(* Logix 5000 project; controller Good_Foods_96985_10252022_1208 vendor 1 type 14 code 151 rev 32.15; software revision 32.04; part 2 of 4 *)
(* tags used below, declared in another part *)
   Active_Container_Recipe : Container_Recipe;
   bAccess_Allowed : BOOL;
   bAccess_Not_Allowed : BOOL;
   bActive_Cleanout_Mode : BOOL;
   bAlwaysOff : BOOL;
   bFault_Active : BOOL;
   bHMI_PB_Left_Denester_Enabled : BOOL;
   bHMI_PB_Left_DropGate_EXT : BOOL;
   bHMI_PB_Left_DropGate_RET : BOOL;
   bHMI_PB_Left_Shuttle_EXT : BOOL;
   bHMI_PB_Left_Shuttle_RET : BOOL;
   bHMI_PB_Load_Recipe : BOOL;
   bHMI_PB_Right_Denester_Enabled : BOOL;
   bHMI_PB_Right_DropGate_EXT : BOOL;
   bHMI_PB_Right_DropGate_RET : BOOL;
   bHMI_PB_Right_Shuttle_EXT : BOOL;
   bHMI_PB_Right_Shuttle_RET : BOOL;
   bHMI_PB_Save_Recipe : BOOL;
   bHmi_PB_Set_Encoder_Home_Position : BOOL;
   bHome_1 : BOOL;
   bHome_Master_Encoder : BOOL;
   bHoming_Cmplt : BOOL;
   bHoming_Step_1 : BOOL;
   bLeft_Indexing : BOOL;
   bLeft_System_Not_Running : BOOL;
   bLeftConvBacklog_OK : BOOL;
   bLeftDropBacklog_OK : BOOL;
   bLeftPrimeBacklog_OK : BOOL;
   bLeftShuttleBacklog_OK : BOOL;
   bMaster_Encoder_Homed_After_Restart : BOOL;
   bRight_Indexing : BOOL;
   bRight_System_Not_Running : BOOL;
   bRightConvBacklog_OK : BOOL;
   bRightDropBacklog_OK : BOOL;
   bRightPrimeBacklog_OK : BOOL;
   bRightShuttleBacklog_OK : BOOL;
   bSystem_Active : BOOL;
   bSystem_Needs_To_Be_Homed : BOOL;
   Cmplt_Homing_Step_1 : BOOL;
   Container_Recipe : Container_Recipe[32];
   ctuInitLeftCyl : COUNTER;
   ctuInitRightCyl : COUNTER;   // Wont Repeat Initilation Sequence If Cmplt
   dAlarms : DINT[8];
   dHoming_Count : DINT;
   DI_PE_Left_Conv_Backlog_Present : BOOL;
   DI_PE_Left_Denest_Prime_OK : BOOL;
   DI_PE_Left_Drop_Cont_Present : BOOL;
   DI_PE_Left_Shuttle_Backlog_Present : BOOL;
   DI_PE_Right_Conv_Backlog_Present : BOOL;
   DI_PE_Right_Denest_Prime_OK : BOOL;
   DI_PE_Right_Drop_Cont_Present : BOOL;
   DI_PE_Right_Shuttle_Backlog_Present : BOOL;
   DI_PRX_Left_DropGate_EXT : BOOL;
   DI_PRX_Left_DropGate_RET : BOOL;
   DI_PRX_Left_Shuttle_RET : BOOL;
   DI_PRX_LugChain_HomingProx : BOOL;
   DI_PRX_Right_DropGate_EXT : BOOL;
   DI_PRX_Right_DropGate_RET : BOOL;
   DI_PRX_Right_Shuttle_RET : BOOL;
   dLeft_Shuttle_Seq_CMD : DINT;
   dLeft_Shuttle_Seq_CMPLT : DINT;
   DO_SOL_Left_DropGate_EXT : BOOL;
   DO_SOL_Left_DropGate_RET : BOOL;
   DO_SOL_Left_Shuttle_EXT : BOOL;
   DO_SOL_Left_Shuttle_RET : BOOL;
   DO_SOL_Right_DropGate_EXT : BOOL;
   DO_SOL_Right_DropGate_RET : BOOL;
   DO_SOL_Right_Shuttle_EXT : BOOL;
   DO_SOL_Right_Shuttle_RET : BOOL;
   dRight_Shuttle_Seq_CMD : DINT;
   dRight_Shuttle_Seq_CMPLT : DINT;
   dSystem_Start_Seq_CMPLT : DINT;
   dSystem_Stop_Seq_CMPLT : DINT;
   intHMI_RecipeListPntr : INT;
   intRecipePntr : INT;
   Left_Rev_Count : INT;
   LugChain_HomingProx_ONS : BOOL;
   LugChain_ONS_Rising : BOOL;
   mamAxisLeftSCREW_INDEXMOVE : MOTION_INSTRUCTION;
   mamAxisRightSCREW_INDEXMOVE : MOTION_INSTRUCTION;
   Master_Encoder : AXIS_CIP_DRIVE;
   ONS : DINT[16];
   rHMI_Drop_Position_Save : REAL;
   rHMI_Index_Speed_Save : REAL;
   rHMI_LefPrime_Backlog_Start_Time_S : REAL;
   rHMI_Left_Denester_Park_Pos_Save : REAL;
   rHMI_LeftConv_Backlog_Start_Time_S : REAL;
   rHMI_LeftConv_Backlog_Stop_Time_S : REAL;
   rHMI_LeftDrop_Backlog_Start_Time_S : REAL;
   rHMI_LeftDrop_Backlog_Stop_Time_S : REAL;
   rHMI_LeftPrime_Backlog_Stop_Time_S : REAL;
   rHMI_LeftShuttle_Backlog_Start_Time_S : REAL;
   rHMI_LeftShuttle_Backlog_Stop_Time_S : REAL;
   rHMI_Right_Denester_Park_Pos_Save : REAL;
   rHMI_RightConv_Backlog_Start_Time_S : REAL;
   rHMI_RightConv_Backlog_Stop_Time_S : REAL;
   rHMI_RightDrop_Backlog_Start_Time_S : REAL;
   rHMI_RightDrop_Backlog_Stop_Time_S : REAL;
   rHMI_RightPrime_Backlog_Start_Time_S : REAL;
   rHMI_RightPrime_Backlog_Stop_Time_S : REAL;
   rHMI_RightShuttle_Backlog_Start_Time_S : REAL;
   rHMI_RightShuttle_Backlog_Stop_Time_S : REAL;
   rHome_Encoder_High_Limit : REAL;
   rHome_Encoder_Low_Limit : REAL;
   Right_Rev_Count : INT;
   rSIKO_Rail_Position_Save : REAL;
   strEmpty_String : STRING;
   strHMI_Current_User : STRING;
   String : STRING;
   strMaint_String : STRING;
   strMCHS_String : STRING;
   tLeftConv_Backlog_Start : TIMER;
   tLeftConv_Backlog_Stop : TIMER;
   tLeftDrop_Backlog_Start : TIMER;
   tLeftDrop_Backlog_Stop : TIMER;
   tLeftExtDrpDly : TIMER;
   tLeftExtShutDly : TIMER;
   tLeftPrime_Backlog_Start : TIMER;
   tLeftPrime_Backlog_Stop : TIMER;
   tLeftRetDrpDly : TIMER;
   tLeftRetShutDly : TIMER;
   tLeftShuttle_Backlog_Start : TIMER;
   tLeftShuttle_Backlog_Stop : TIMER;
   tRightConv_Backlog_Start : TIMER;
   tRightConv_Backlog_Stop : TIMER;
   tRightDrop_Backlog_Start : TIMER;
   tRightDrop_Backlog_Stop : TIMER;
   tRightExtDrpDly : TIMER;
   tRightExtShutDly : TIMER;
   tRightPrime_Backlog_Start : TIMER;
   tRightPrime_Backlog_Stop : TIMER;
   tRightRetDrpDly : TIMER;
   tRightRetShutDly : TIMER;
   tRightShuttle_Backlog_Start : TIMER;
   tRightShuttle_Backlog_Stop : TIMER;
   tRightStopPosDly : TIMER;
   tRightStopPosTimeOut : TIMER;
   tTimer_Homing : TIMER;
(* MainProgram, continued *)

ROUTINE _11_Left_Shuttle_Control   (* ladder *)
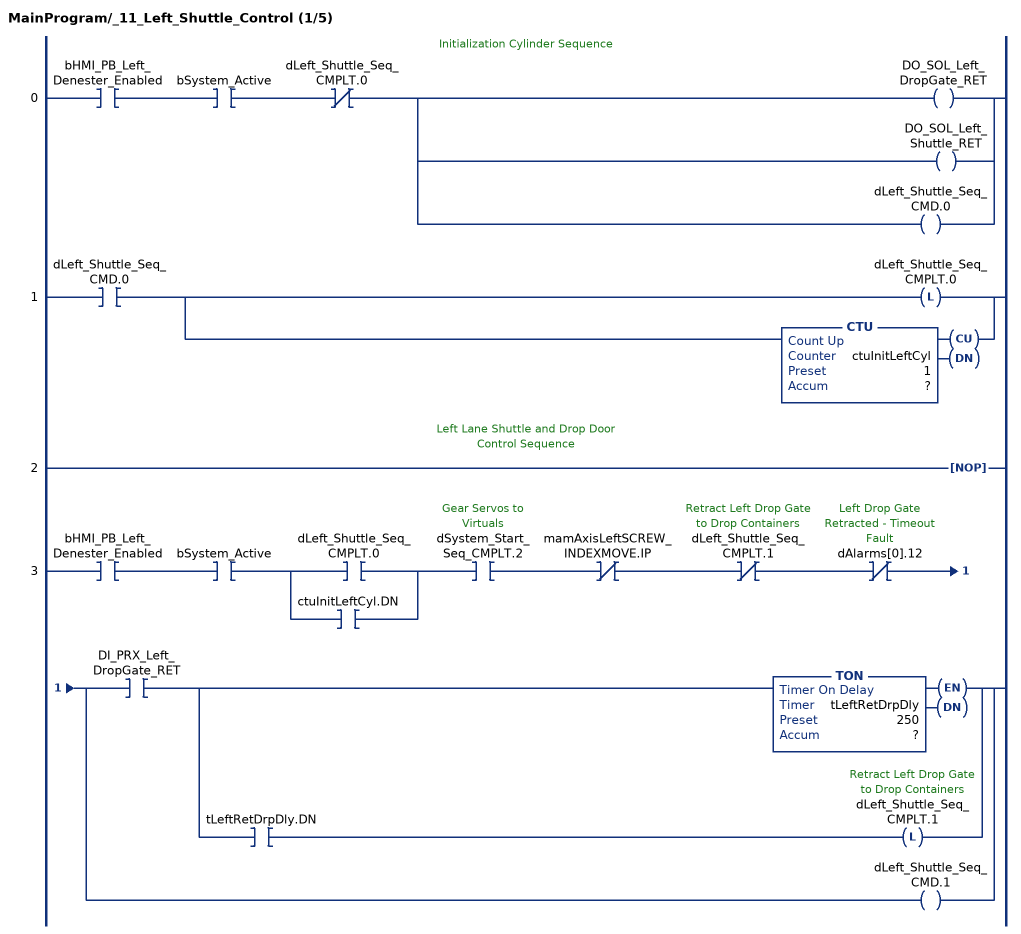
   // Initialization Cylinder Sequence
   0: XIC(bHMI_PB_Left_Denester_Enabled)XIC(bSystem_Active)XIO(dLeft_Shuttle_Seq_CMPLT.0)[OTE(DO_SOL_Left_DropGate_RET) ,OTE(DO_SOL_Left_Shuttle_RET) ,OTE(dLeft_Shuttle_Seq_CMD.0) ];
   1: XIC(dLeft_Shuttle_Seq_CMD.0)[OTL(dLeft_Shuttle_Seq_CMPLT.0) ,CTU(ctuInitLeftCyl,?,?) ];
   // Left Lane Shuttle and Drop Door
   // Control Sequence
   2: NOP();
   3: XIC(bHMI_PB_Left_Denester_Enabled)XIC(bSystem_Active)[XIC(dLeft_Shuttle_Seq_CMPLT.0) ,XIC(ctuInitLeftCyl.DN) ]XIC(dSystem_Start_Seq_CMPLT.2)XIO(mamAxisLeftSCREW_INDEXMOVE.IP)XIO(dLeft_Shuttle_Seq_CMPLT.1)XIO(dAlarms[0].12)[XIC(DI_PRX_Left_DropGate_RET) [TON(tLeftRetDrpDly,?,?) ,XIC(tLeftRetDrpDly.DN) OTL(dLeft_Shuttle_Seq_CMPLT.1) ] ,OTE(dLeft_Shuttle_Seq_CMD.1) ];
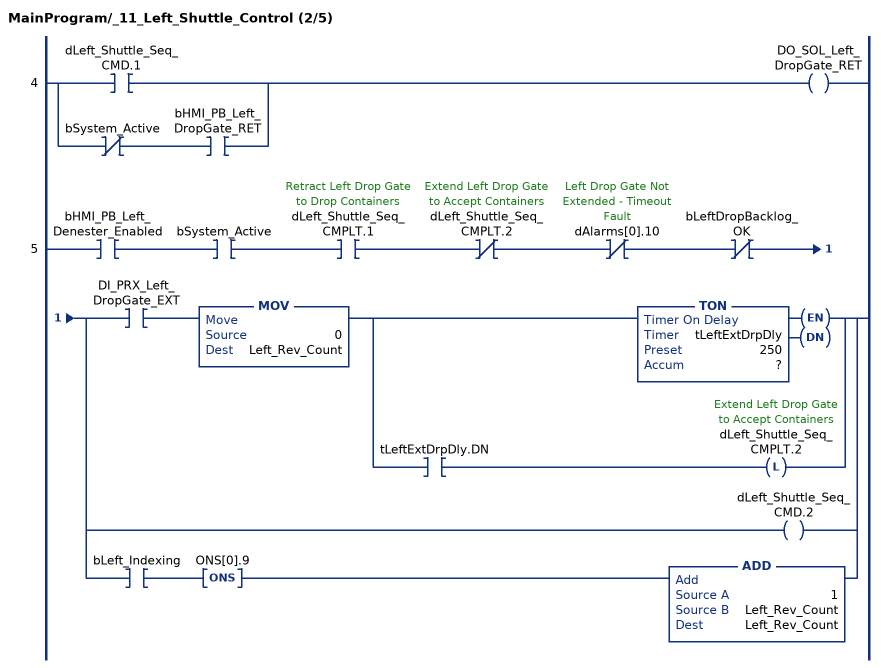
   4: [XIC(dLeft_Shuttle_Seq_CMD.1) ,XIO(bSystem_Active) XIC(bHMI_PB_Left_DropGate_RET) ]OTE(DO_SOL_Left_DropGate_RET);
   5: XIC(bHMI_PB_Left_Denester_Enabled)XIC(bSystem_Active)XIC(dLeft_Shuttle_Seq_CMPLT.1)XIO(dLeft_Shuttle_Seq_CMPLT.2)XIO(dAlarms[0].10)XIO(bLeftDropBacklog_OK)[XIC(DI_PRX_Left_DropGate_EXT) MOV(0,Left_Rev_Count) [TON(tLeftExtDrpDly,?,?) ,XIC(tLeftExtDrpDly.DN) OTL(dLeft_Shuttle_Seq_CMPLT.2) ] ,OTE(dLeft_Shuttle_Seq_CMD.2) ,XIC(bLeft_Indexing) ONS(ONS[0].9) ADD(1,Left_Rev_Count,Left_Rev_Count) ];
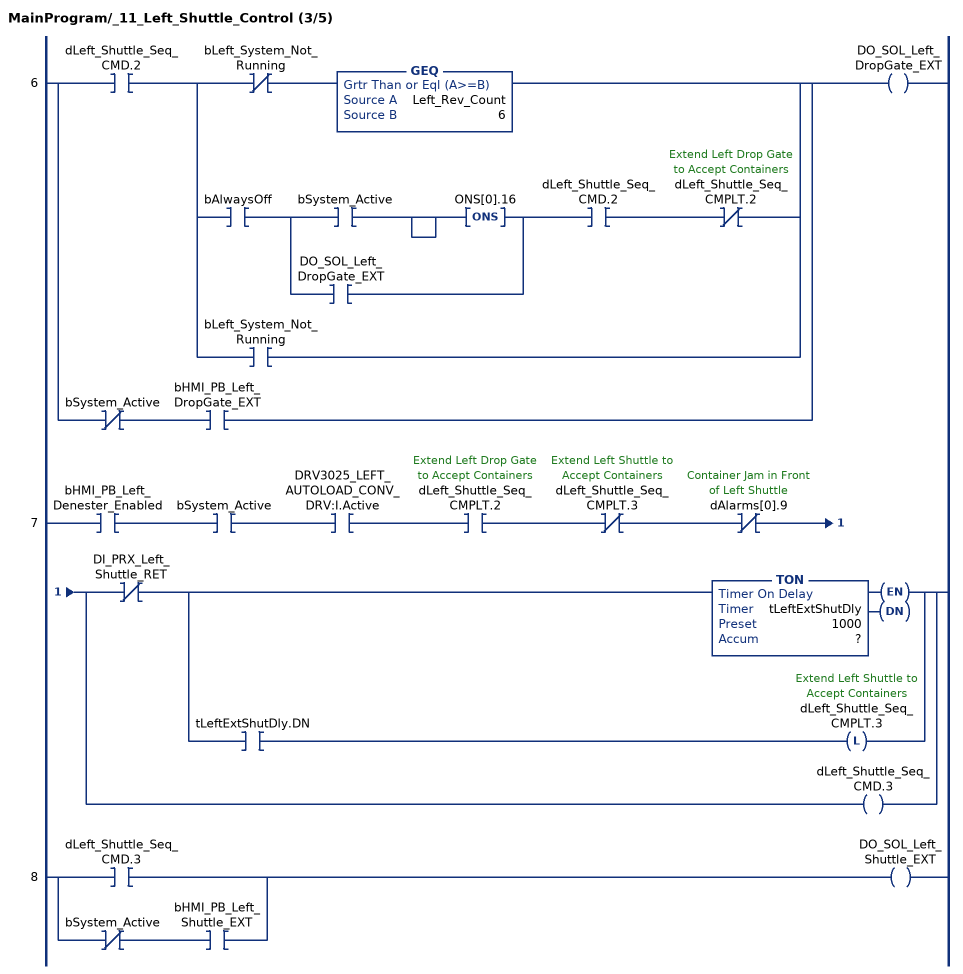
   6: [XIC(dLeft_Shuttle_Seq_CMD.2) [XIO(bLeft_System_Not_Running) GEQ(Left_Rev_Count,6) ,XIC(bAlwaysOff) [XIC(bSystem_Active) [,] ONS(ONS[0].16) ,XIC(DO_SOL_Left_DropGate_EXT) ] XIC(dLeft_Shuttle_Seq_CMD.2) XIO(dLeft_Shuttle_Seq_CMPLT.2) ,XIC(bLeft_System_Not_Running) ] ,XIO(bSystem_Active) XIC(bHMI_PB_Left_DropGate_EXT) ]OTE(DO_SOL_Left_DropGate_EXT);
   7: XIC(bHMI_PB_Left_Denester_Enabled)XIC(bSystem_Active)XIC(DRV3025_LEFT_AUTOLOAD_CONV_DRV:I.Active)XIC(dLeft_Shuttle_Seq_CMPLT.2)XIO(dLeft_Shuttle_Seq_CMPLT.3)XIO(dAlarms[0].9)[XIO(DI_PRX_Left_Shuttle_RET) [TON(tLeftExtShutDly,?,?) ,XIC(tLeftExtShutDly.DN) OTL(dLeft_Shuttle_Seq_CMPLT.3) ] ,OTE(dLeft_Shuttle_Seq_CMD.3) ];
   8: [XIC(dLeft_Shuttle_Seq_CMD.3) ,XIO(bSystem_Active) XIC(bHMI_PB_Left_Shuttle_EXT) ]OTE(DO_SOL_Left_Shuttle_EXT);
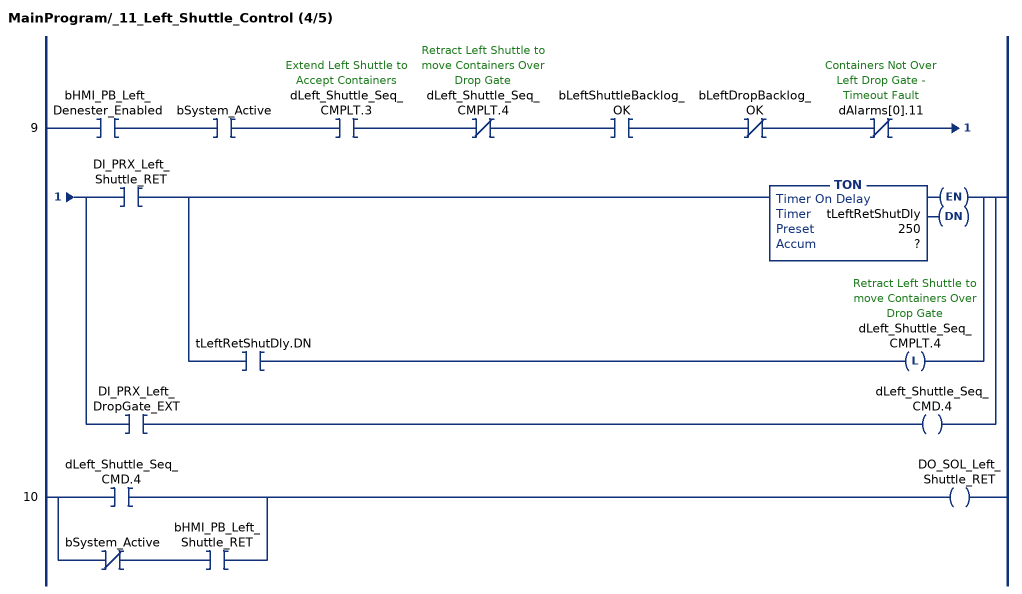
   9: XIC(bHMI_PB_Left_Denester_Enabled)XIC(bSystem_Active)XIC(dLeft_Shuttle_Seq_CMPLT.3)XIO(dLeft_Shuttle_Seq_CMPLT.4)XIC(bLeftShuttleBacklog_OK)XIO(bLeftDropBacklog_OK)XIO(dAlarms[0].11)[XIC(DI_PRX_Left_Shuttle_RET) [TON(tLeftRetShutDly,?,?) ,XIC(tLeftRetShutDly.DN) OTL(dLeft_Shuttle_Seq_CMPLT.4) ] ,XIC(DI_PRX_Left_DropGate_EXT) OTE(dLeft_Shuttle_Seq_CMD.4) ];
   10: [XIC(dLeft_Shuttle_Seq_CMD.4) ,XIO(bSystem_Active) XIC(bHMI_PB_Left_Shuttle_RET) ]OTE(DO_SOL_Left_Shuttle_RET);
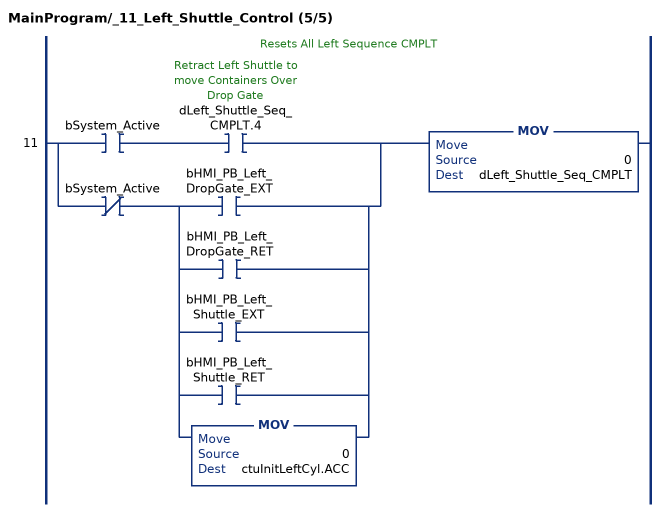
   // Resets All Left Sequence CMPLT
   11: [XIC(bSystem_Active) XIC(dLeft_Shuttle_Seq_CMPLT.4) ,XIO(bSystem_Active) [XIC(bHMI_PB_Left_DropGate_EXT) ,XIC(bHMI_PB_Left_DropGate_RET) ,XIC(bHMI_PB_Left_Shuttle_EXT) ,XIC(bHMI_PB_Left_Shuttle_RET) ,MOV(0,ctuInitLeftCyl.ACC) ] ]MOV(0,dLeft_Shuttle_Seq_CMPLT);
END_ROUTINE

ROUTINE _12_Right_Shuttle_Control   (* ladder *)
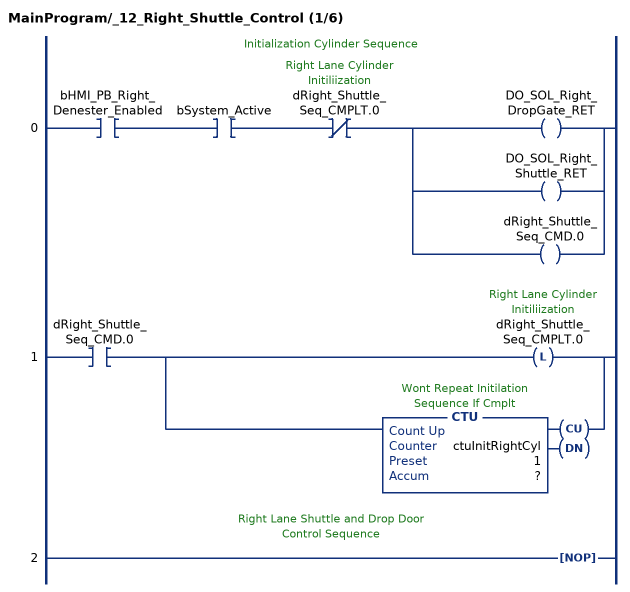
   // Initialization Cylinder Sequence
   0: XIC(bHMI_PB_Right_Denester_Enabled)XIC(bSystem_Active)XIO(dRight_Shuttle_Seq_CMPLT.0)[OTE(DO_SOL_Right_DropGate_RET) ,OTE(DO_SOL_Right_Shuttle_RET) ,OTE(dRight_Shuttle_Seq_CMD.0) ];
   1: XIC(dRight_Shuttle_Seq_CMD.0)[OTL(dRight_Shuttle_Seq_CMPLT.0) ,CTU(ctuInitRightCyl,?,?) ];
   // Right Lane Shuttle and Drop Door
   // Control Sequence
   2: NOP();
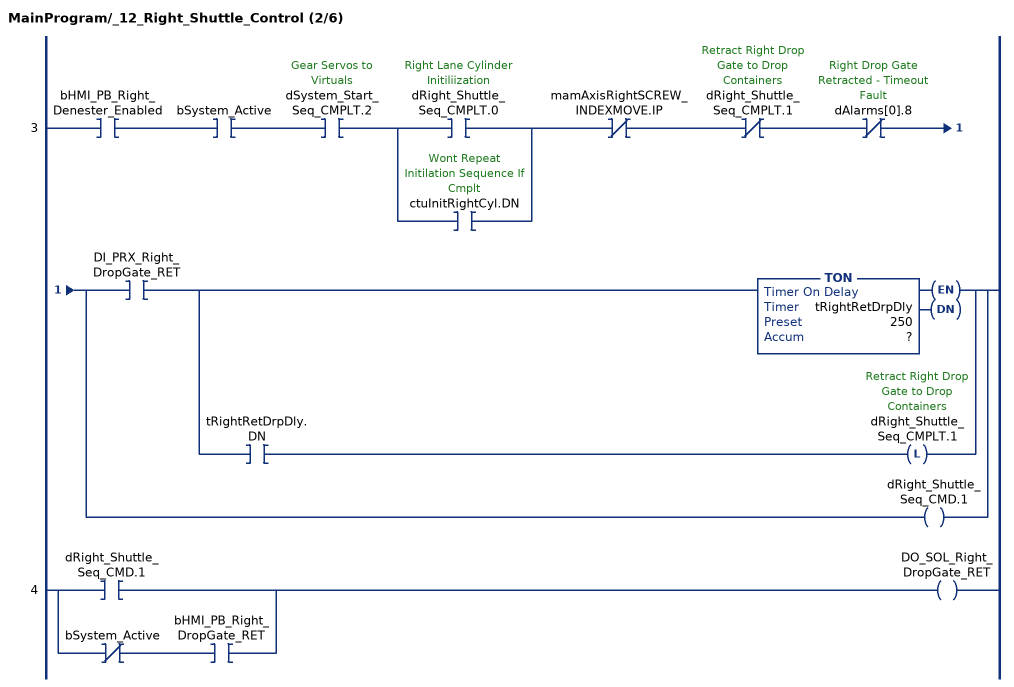
   3: XIC(bHMI_PB_Right_Denester_Enabled)XIC(bSystem_Active)XIC(dSystem_Start_Seq_CMPLT.2)[XIC(dRight_Shuttle_Seq_CMPLT.0) ,XIC(ctuInitRightCyl.DN) ]XIO(mamAxisRightSCREW_INDEXMOVE.IP)XIO(dRight_Shuttle_Seq_CMPLT.1)XIO(dAlarms[0].8)[XIC(DI_PRX_Right_DropGate_RET) [TON(tRightRetDrpDly,?,?) ,XIC(tRightRetDrpDly.DN) OTL(dRight_Shuttle_Seq_CMPLT.1) ] ,OTE(dRight_Shuttle_Seq_CMD.1) ];
   4: [XIC(dRight_Shuttle_Seq_CMD.1) ,XIO(bSystem_Active) XIC(bHMI_PB_Right_DropGate_RET) ]OTE(DO_SOL_Right_DropGate_RET);
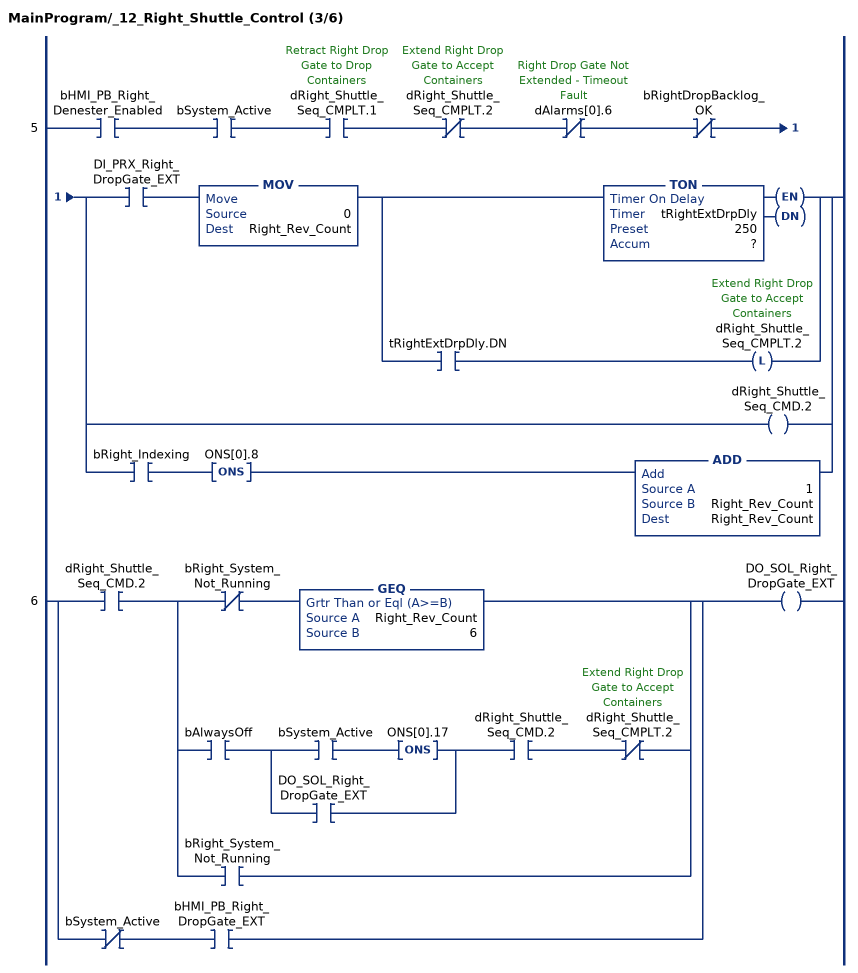
   5: XIC(bHMI_PB_Right_Denester_Enabled)XIC(bSystem_Active)XIC(dRight_Shuttle_Seq_CMPLT.1)XIO(dRight_Shuttle_Seq_CMPLT.2)XIO(dAlarms[0].6)XIO(bRightDropBacklog_OK)[XIC(DI_PRX_Right_DropGate_EXT) MOV(0,Right_Rev_Count) [TON(tRightExtDrpDly,?,?) ,XIC(tRightExtDrpDly.DN) OTL(dRight_Shuttle_Seq_CMPLT.2) ] ,OTE(dRight_Shuttle_Seq_CMD.2) ,XIC(bRight_Indexing) ONS(ONS[0].8) ADD(1,Right_Rev_Count,Right_Rev_Count) ];
   6: [XIC(dRight_Shuttle_Seq_CMD.2) [XIO(bRight_System_Not_Running) GEQ(Right_Rev_Count,6) ,XIC(bAlwaysOff) [XIC(bSystem_Active) ONS(ONS[0].17) ,XIC(DO_SOL_Right_DropGate_EXT) ] XIC(dRight_Shuttle_Seq_CMD.2) XIO(dRight_Shuttle_Seq_CMPLT.2) ,XIC(bRight_System_Not_Running) ] ,XIO(bSystem_Active) XIC(bHMI_PB_Right_DropGate_EXT) ]OTE(DO_SOL_Right_DropGate_EXT);
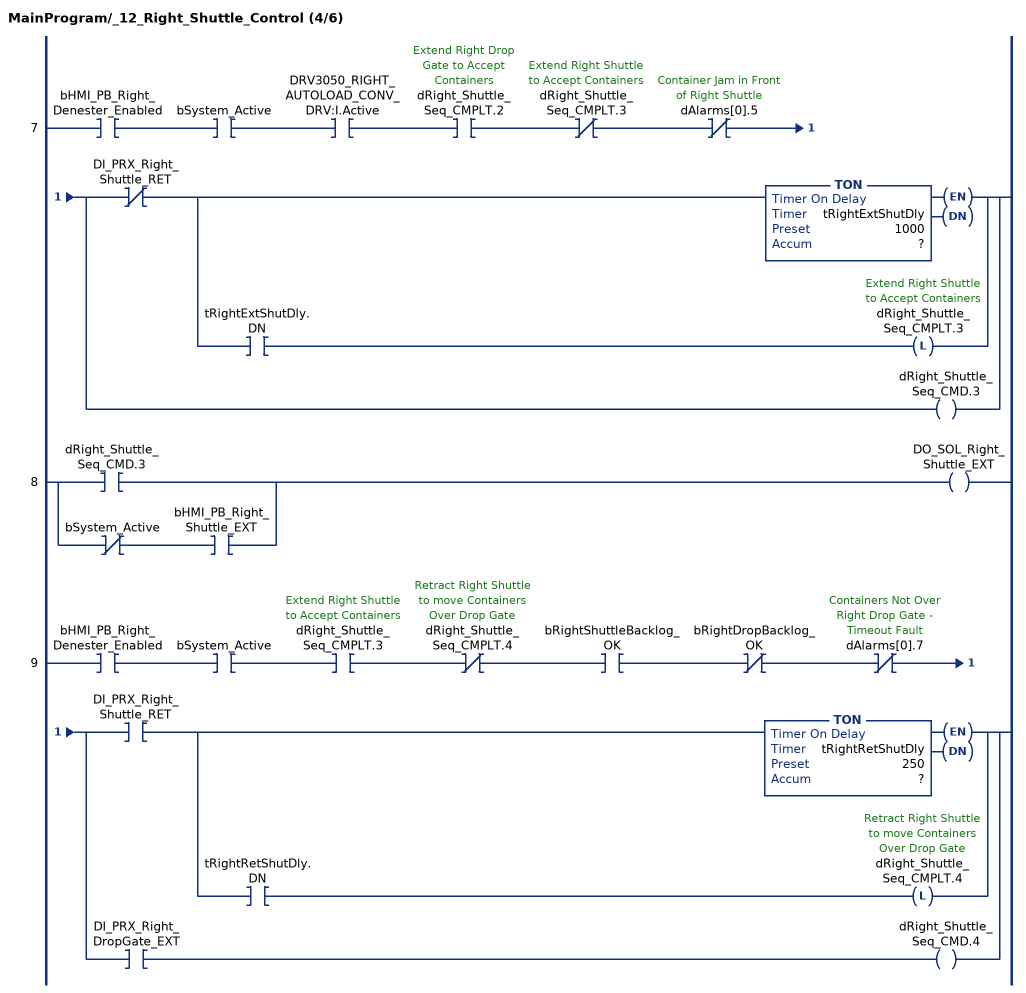
   7: XIC(bHMI_PB_Right_Denester_Enabled)XIC(bSystem_Active)XIC(DRV3050_RIGHT_AUTOLOAD_CONV_DRV:I.Active)XIC(dRight_Shuttle_Seq_CMPLT.2)XIO(dRight_Shuttle_Seq_CMPLT.3)XIO(dAlarms[0].5)[XIO(DI_PRX_Right_Shuttle_RET) [TON(tRightExtShutDly,?,?) ,XIC(tRightExtShutDly.DN) OTL(dRight_Shuttle_Seq_CMPLT.3) ] ,OTE(dRight_Shuttle_Seq_CMD.3) ];
   8: [XIC(dRight_Shuttle_Seq_CMD.3) ,XIO(bSystem_Active) XIC(bHMI_PB_Right_Shuttle_EXT) ]OTE(DO_SOL_Right_Shuttle_EXT);
   9: XIC(bHMI_PB_Right_Denester_Enabled)XIC(bSystem_Active)XIC(dRight_Shuttle_Seq_CMPLT.3)XIO(dRight_Shuttle_Seq_CMPLT.4)XIC(bRightShuttleBacklog_OK)XIO(bRightDropBacklog_OK)XIO(dAlarms[0].7)[XIC(DI_PRX_Right_Shuttle_RET) [TON(tRightRetShutDly,?,?) ,XIC(tRightRetShutDly.DN) OTL(dRight_Shuttle_Seq_CMPLT.4) ] ,XIC(DI_PRX_Right_DropGate_EXT) OTE(dRight_Shuttle_Seq_CMD.4) ];
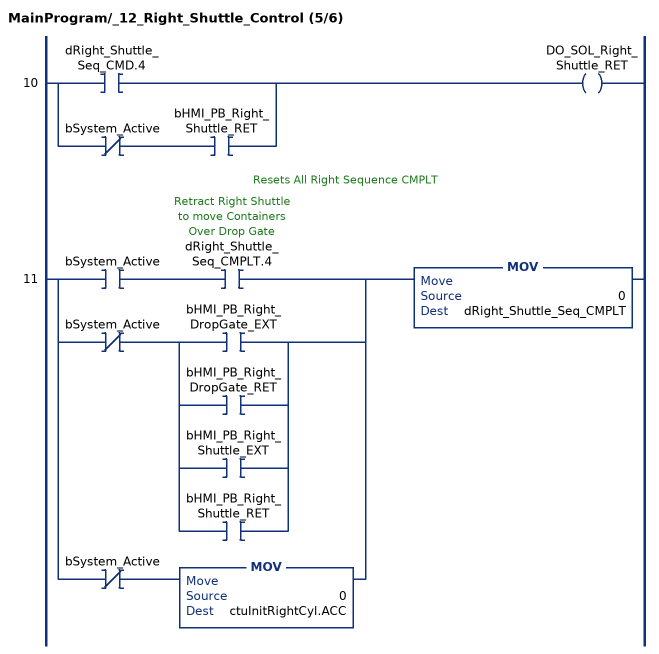
   10: [XIC(dRight_Shuttle_Seq_CMD.4) ,XIO(bSystem_Active) XIC(bHMI_PB_Right_Shuttle_RET) ]OTE(DO_SOL_Right_Shuttle_RET);
   // Resets All Right Sequence CMPLT
   11: [XIC(bSystem_Active) XIC(dRight_Shuttle_Seq_CMPLT.4) ,XIO(bSystem_Active) [XIC(bHMI_PB_Right_DropGate_EXT) ,XIC(bHMI_PB_Right_DropGate_RET) ,XIC(bHMI_PB_Right_Shuttle_EXT) ,XIC(bHMI_PB_Right_Shuttle_RET) ] ,XIO(bSystem_Active) MOV(0,ctuInitRightCyl.ACC) ]MOV(0,dRight_Shuttle_Seq_CMPLT);
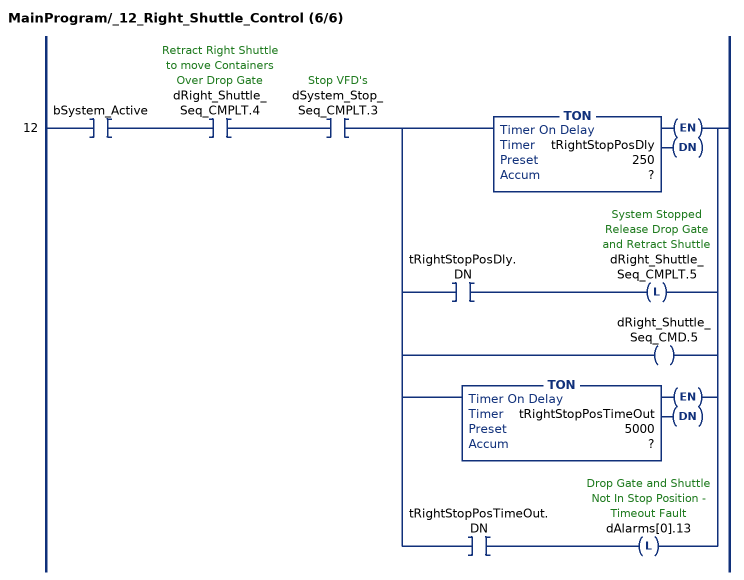
   12: XIC(bSystem_Active)XIC(dRight_Shuttle_Seq_CMPLT.4)XIC(dSystem_Stop_Seq_CMPLT.3)[TON(tRightStopPosDly,?,?) ,XIC(tRightStopPosDly.DN) OTL(dRight_Shuttle_Seq_CMPLT.5) ,OTE(dRight_Shuttle_Seq_CMD.5) ,TON(tRightStopPosTimeOut,?,?) ,XIC(tRightStopPosTimeOut.DN) OTL(dAlarms[0].13) ];
END_ROUTINE

ROUTINE _13_Recipe   (* ladder *)
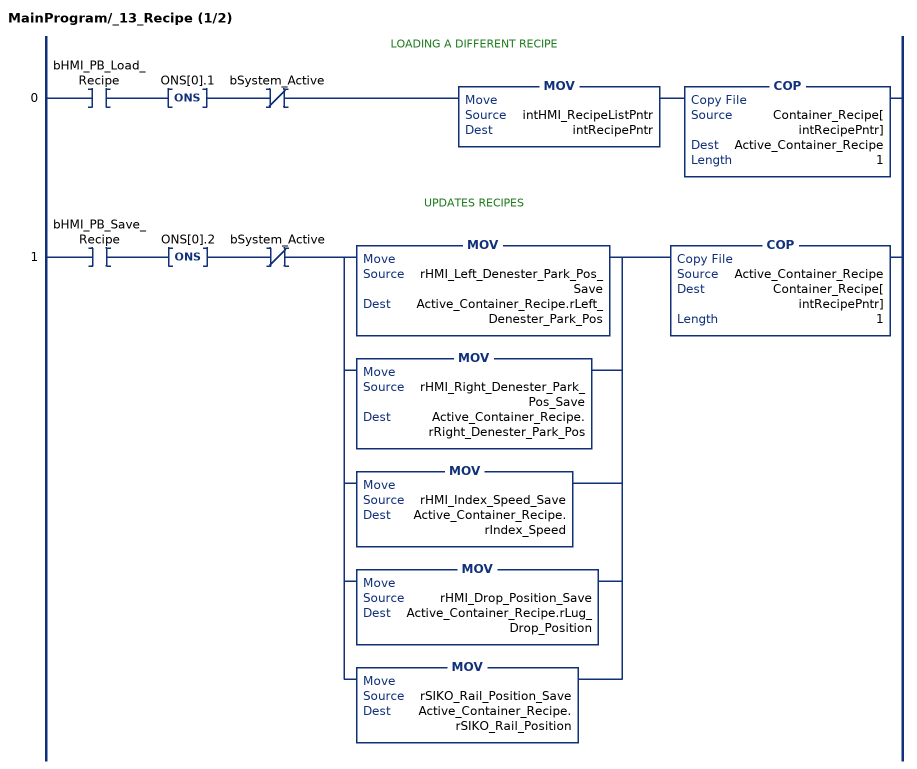
   // LOADING A DIFFERENT RECIPE
   0: XIC(bHMI_PB_Load_Recipe)ONS(ONS[0].1)XIO(bSystem_Active)MOV(intHMI_RecipeListPntr,intRecipePntr)COP(Container_Recipe[intRecipePntr],Active_Container_Recipe,1);
   // UPDATES RECIPES
   1: XIC(bHMI_PB_Save_Recipe)ONS(ONS[0].2)XIO(bSystem_Active)[MOV(rHMI_Left_Denester_Park_Pos_Save,Active_Container_Recipe.rLeft_Denester_Park_Pos) ,MOV(rHMI_Right_Denester_Park_Pos_Save,Active_Container_Recipe.rRight_Denester_Park_Pos) ,MOV(rHMI_Index_Speed_Save,Active_Container_Recipe.rIndex_Speed) ,MOV(rHMI_Drop_Position_Save,Active_Container_Recipe.rLug_Drop_Position) ,MOV(rSIKO_Rail_Position_Save,Active_Container_Recipe.rSIKO_Rail_Position) ]COP(Active_Container_Recipe,Container_Recipe[intRecipePntr],1);
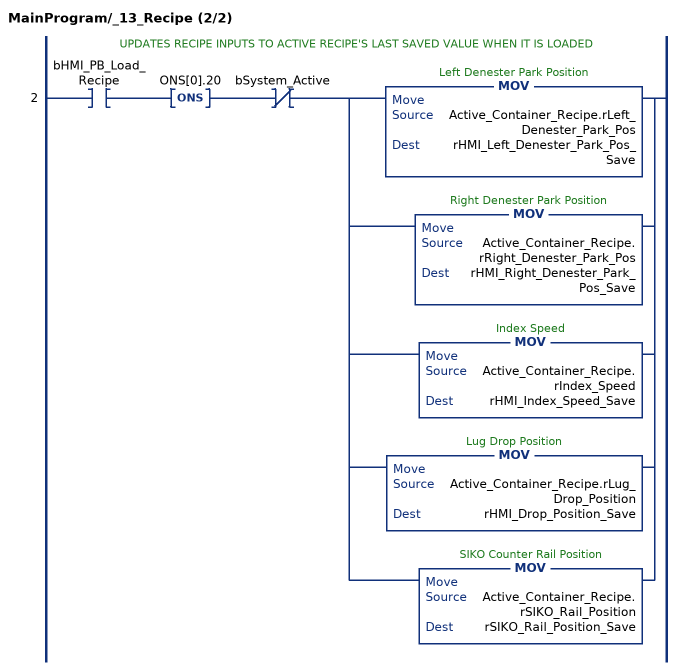
   // UPDATES RECIPE INPUTS TO ACTIVE RECIPE'S LAST SAVED VALUE WHEN IT IS LOADED
   2: XIC(bHMI_PB_Load_Recipe)ONS(ONS[0].20)XIO(bSystem_Active)[MOV(Active_Container_Recipe.rLeft_Denester_Park_Pos,rHMI_Left_Denester_Park_Pos_Save) ,MOV(Active_Container_Recipe.rRight_Denester_Park_Pos,rHMI_Right_Denester_Park_Pos_Save) ,MOV(Active_Container_Recipe.rIndex_Speed,rHMI_Index_Speed_Save) ,MOV(Active_Container_Recipe.rLug_Drop_Position,rHMI_Drop_Position_Save) ,MOV(Active_Container_Recipe.rSIKO_Rail_Position,rSIKO_Rail_Position_Save) ];
END_ROUTINE

ROUTINE _14_Home_Encoder   (* ladder *)
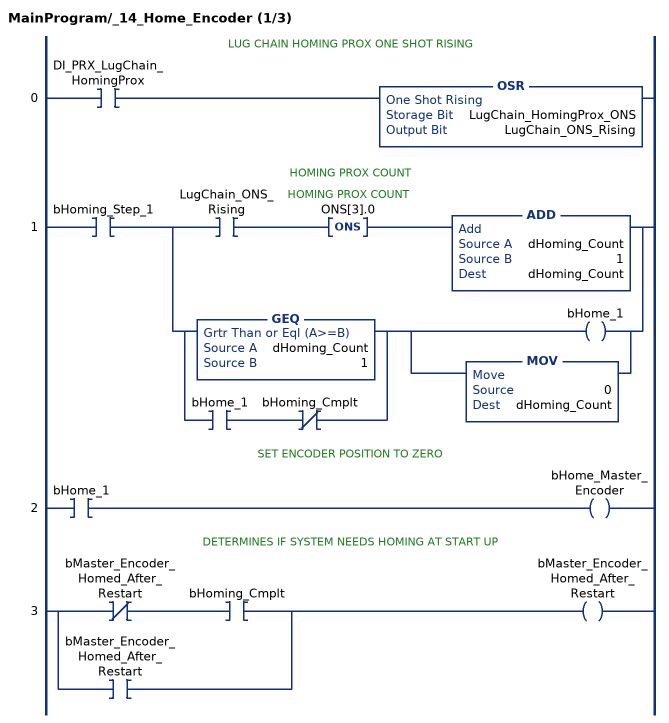
   // LUG CHAIN HOMING PROX ONE SHOT RISING
   0: XIC(DI_PRX_LugChain_HomingProx)OSR(LugChain_HomingProx_ONS,LugChain_ONS_Rising);
   // HOMING PROX COUNT
   1: XIC(bHoming_Step_1)[XIC(LugChain_ONS_Rising) ONS(ONS[3].0) ADD(dHoming_Count,1,dHoming_Count) ,[GEQ(dHoming_Count,1) ,XIC(bHome_1) XIO(bHoming_Cmplt) ] [OTE(bHome_1) ,MOV(0,dHoming_Count) ] ];
   // SET ENCODER POSITION TO ZERO
   2: XIC(bHome_1)OTE(bHome_Master_Encoder);
   // DETERMINES IF SYSTEM NEEDS HOMING AT START UP
   3: [XIO(bMaster_Encoder_Homed_After_Restart) XIC(bHoming_Cmplt) ,XIC(bMaster_Encoder_Homed_After_Restart) ]OTE(bMaster_Encoder_Homed_After_Restart);
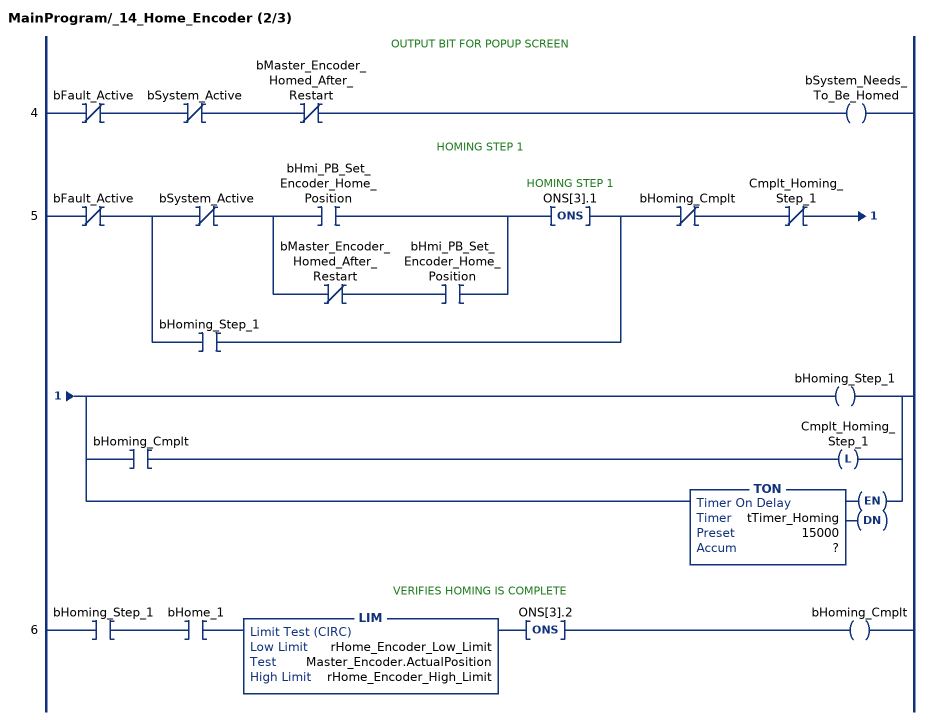
   // OUTPUT BIT FOR POPUP SCREEN
   4: XIO(bFault_Active)XIO(bSystem_Active)XIO(bMaster_Encoder_Homed_After_Restart)OTE(bSystem_Needs_To_Be_Homed);
   // HOMING STEP 1
   5: XIO(bFault_Active)[XIO(bSystem_Active) [XIC(bHmi_PB_Set_Encoder_Home_Position) ,XIO(bMaster_Encoder_Homed_After_Restart) XIC(bHmi_PB_Set_Encoder_Home_Position) ] ONS(ONS[3].1) ,XIC(bHoming_Step_1) ]XIO(bHoming_Cmplt)XIO(Cmplt_Homing_Step_1)[OTE(bHoming_Step_1) ,XIC(bHoming_Cmplt) OTL(Cmplt_Homing_Step_1) ,TON(tTimer_Homing,?,?) ];
   // VERIFIES HOMING IS COMPLETE
   6: XIC(bHoming_Step_1)XIC(bHome_1)LIM(rHome_Encoder_Low_Limit,Master_Encoder.ActualPosition,rHome_Encoder_High_Limit)ONS(ONS[3].2)OTE(bHoming_Cmplt);
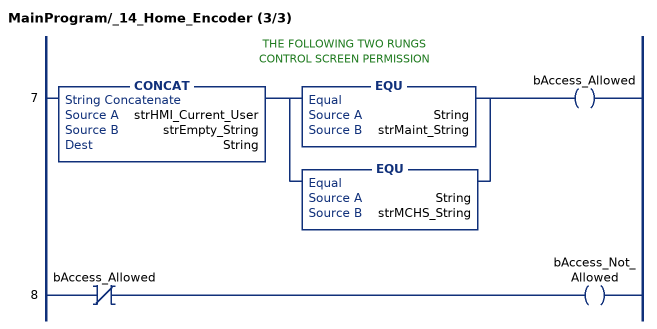
   // THE FOLLOWING TWO RUNGS
   // CONTROL SCREEN PERMISSION
   7: CONCAT(strHMI_Current_User,strEmpty_String,String)[EQU(String,strMaint_String) ,EQU(String,strMCHS_String) ]OTE(bAccess_Allowed);
   8: XIO(bAccess_Allowed)OTE(bAccess_Not_Allowed);
END_ROUTINE

ROUTINE _15_Backlog   (* ladder *)
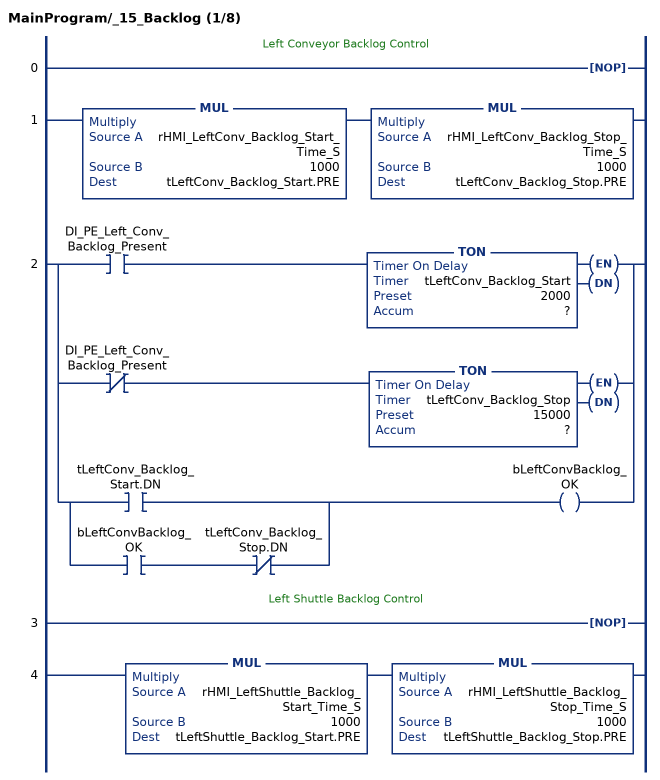
   // Left Conveyor Backlog Control
   0: NOP();
   1: MUL(rHMI_LeftConv_Backlog_Start_Time_S,1000,tLeftConv_Backlog_Start.PRE)MUL(rHMI_LeftConv_Backlog_Stop_Time_S,1000,tLeftConv_Backlog_Stop.PRE);
   2: [XIC(DI_PE_Left_Conv_Backlog_Present) TON(tLeftConv_Backlog_Start,?,?) ,XIO(DI_PE_Left_Conv_Backlog_Present) TON(tLeftConv_Backlog_Stop,?,?) ,[XIC(tLeftConv_Backlog_Start.DN) ,XIC(bLeftConvBacklog_OK) XIO(tLeftConv_Backlog_Stop.DN) ] OTE(bLeftConvBacklog_OK) ];
   // Left Shuttle Backlog Control
   3: NOP();
   4: MUL(rHMI_LeftShuttle_Backlog_Start_Time_S,1000,tLeftShuttle_Backlog_Start.PRE)MUL(rHMI_LeftShuttle_Backlog_Stop_Time_S,1000,tLeftShuttle_Backlog_Stop.PRE);
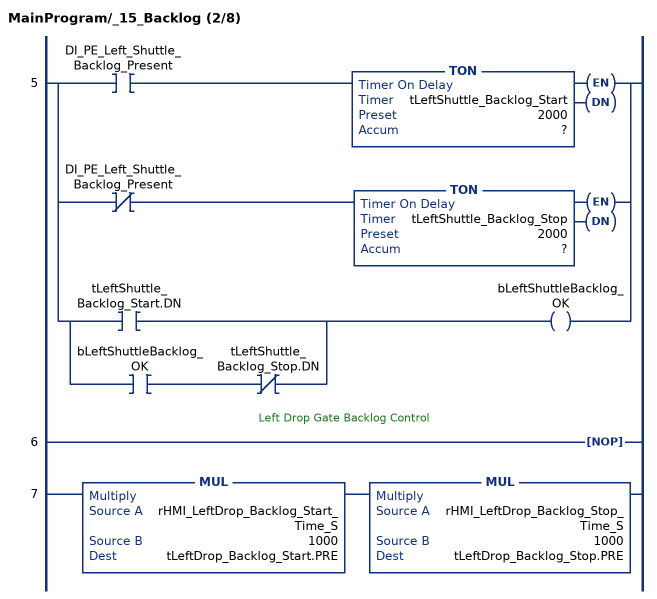
   5: [XIC(DI_PE_Left_Shuttle_Backlog_Present) TON(tLeftShuttle_Backlog_Start,?,?) ,XIO(DI_PE_Left_Shuttle_Backlog_Present) TON(tLeftShuttle_Backlog_Stop,?,?) ,[XIC(tLeftShuttle_Backlog_Start.DN) ,XIC(bLeftShuttleBacklog_OK) XIO(tLeftShuttle_Backlog_Stop.DN) ] OTE(bLeftShuttleBacklog_OK) ];
   // Left Drop Gate Backlog Control
   6: NOP();
   7: MUL(rHMI_LeftDrop_Backlog_Start_Time_S,1000,tLeftDrop_Backlog_Start.PRE)MUL(rHMI_LeftDrop_Backlog_Stop_Time_S,1000,tLeftDrop_Backlog_Stop.PRE);
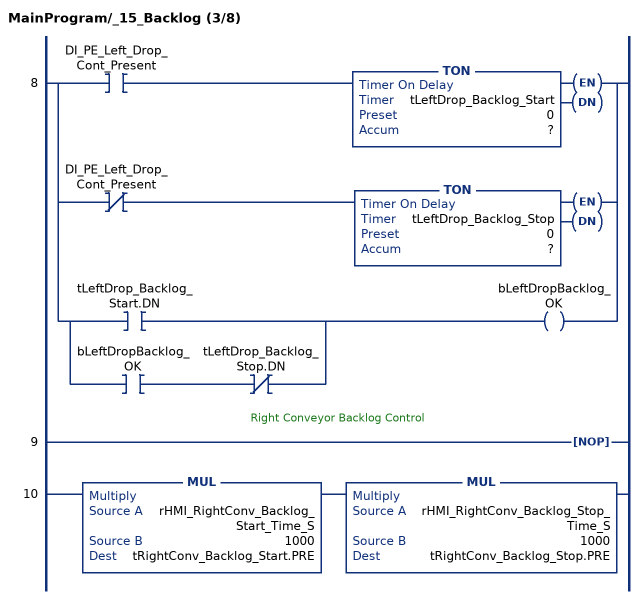
   8: [XIC(DI_PE_Left_Drop_Cont_Present) TON(tLeftDrop_Backlog_Start,?,?) ,XIO(DI_PE_Left_Drop_Cont_Present) TON(tLeftDrop_Backlog_Stop,?,?) ,[XIC(tLeftDrop_Backlog_Start.DN) ,XIC(bLeftDropBacklog_OK) XIO(tLeftDrop_Backlog_Stop.DN) ] OTE(bLeftDropBacklog_OK) ];
   // Right Conveyor Backlog Control
   9: NOP();
   10: MUL(rHMI_RightConv_Backlog_Start_Time_S,1000,tRightConv_Backlog_Start.PRE)MUL(rHMI_RightConv_Backlog_Stop_Time_S,1000,tRightConv_Backlog_Stop.PRE);
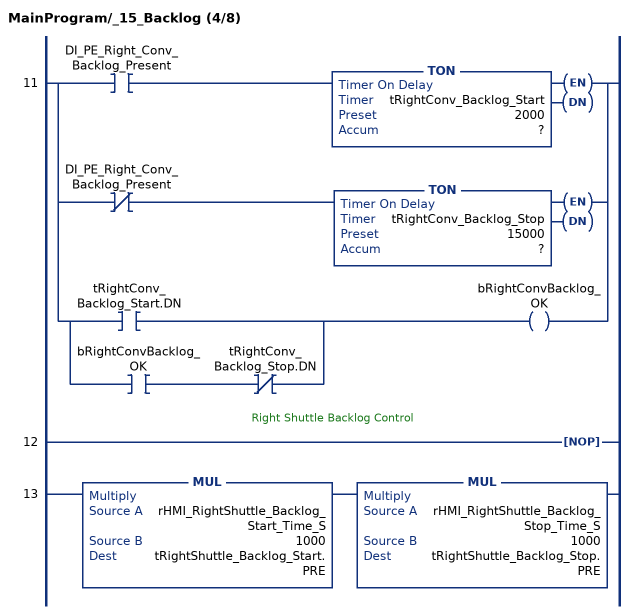
   11: [XIC(DI_PE_Right_Conv_Backlog_Present) TON(tRightConv_Backlog_Start,?,?) ,XIO(DI_PE_Right_Conv_Backlog_Present) TON(tRightConv_Backlog_Stop,?,?) ,[XIC(tRightConv_Backlog_Start.DN) ,XIC(bRightConvBacklog_OK) XIO(tRightConv_Backlog_Stop.DN) ] OTE(bRightConvBacklog_OK) ];
   // Right Shuttle Backlog Control
   12: NOP();
   13: MUL(rHMI_RightShuttle_Backlog_Start_Time_S,1000,tRightShuttle_Backlog_Start.PRE)MUL(rHMI_RightShuttle_Backlog_Stop_Time_S,1000,tRightShuttle_Backlog_Stop.PRE);
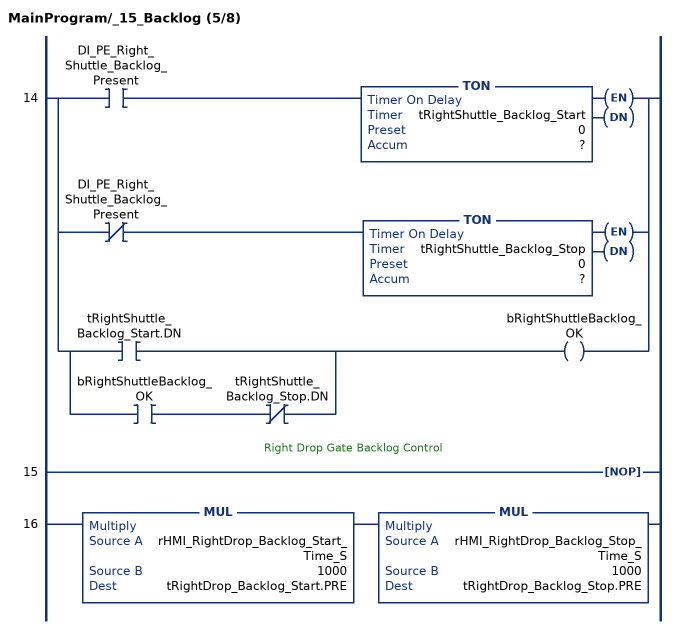
   14: [XIC(DI_PE_Right_Shuttle_Backlog_Present) TON(tRightShuttle_Backlog_Start,?,?) ,XIO(DI_PE_Right_Shuttle_Backlog_Present) TON(tRightShuttle_Backlog_Stop,?,?) ,[XIC(tRightShuttle_Backlog_Start.DN) ,XIC(bRightShuttleBacklog_OK) XIO(tRightShuttle_Backlog_Stop.DN) ] OTE(bRightShuttleBacklog_OK) ];
   // Right Drop Gate Backlog Control
   15: NOP();
   16: MUL(rHMI_RightDrop_Backlog_Start_Time_S,1000,tRightDrop_Backlog_Start.PRE)MUL(rHMI_RightDrop_Backlog_Stop_Time_S,1000,tRightDrop_Backlog_Stop.PRE);
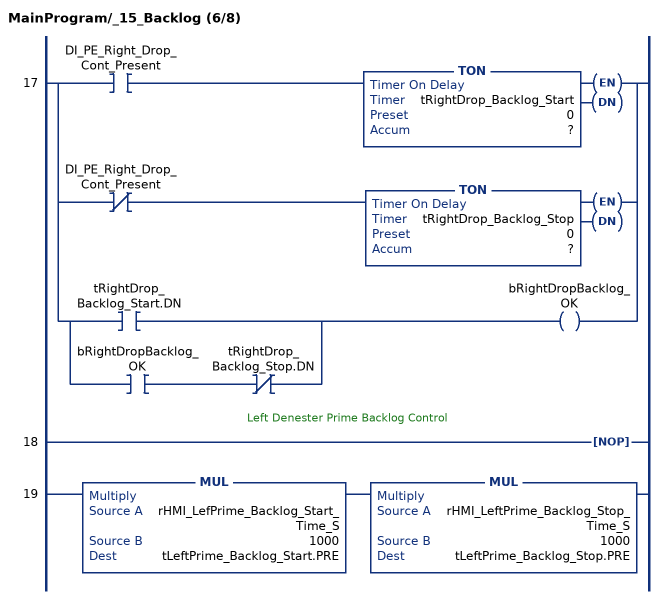
   17: [XIC(DI_PE_Right_Drop_Cont_Present) TON(tRightDrop_Backlog_Start,?,?) ,XIO(DI_PE_Right_Drop_Cont_Present) TON(tRightDrop_Backlog_Stop,?,?) ,[XIC(tRightDrop_Backlog_Start.DN) ,XIC(bRightDropBacklog_OK) XIO(tRightDrop_Backlog_Stop.DN) ] OTE(bRightDropBacklog_OK) ];
   // Left Denester Prime Backlog Control
   18: NOP();
   19: MUL(rHMI_LefPrime_Backlog_Start_Time_S,1000,tLeftPrime_Backlog_Start.PRE)MUL(rHMI_LeftPrime_Backlog_Stop_Time_S,1000,tLeftPrime_Backlog_Stop.PRE);
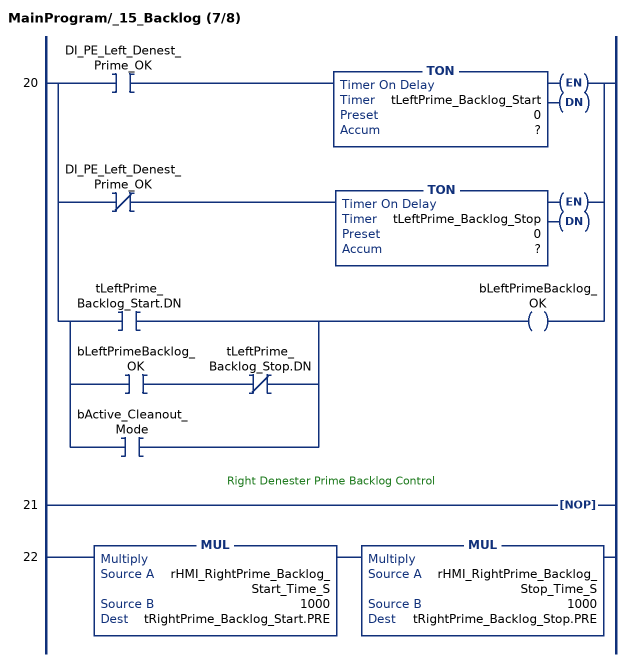
   20: [XIC(DI_PE_Left_Denest_Prime_OK) TON(tLeftPrime_Backlog_Start,?,?) ,XIO(DI_PE_Left_Denest_Prime_OK) TON(tLeftPrime_Backlog_Stop,?,?) ,[XIC(tLeftPrime_Backlog_Start.DN) ,XIC(bLeftPrimeBacklog_OK) XIO(tLeftPrime_Backlog_Stop.DN) ,XIC(bActive_Cleanout_Mode) ] OTE(bLeftPrimeBacklog_OK) ];
   // Right Denester Prime Backlog Control
   21: NOP();
   22: MUL(rHMI_RightPrime_Backlog_Start_Time_S,1000,tRightPrime_Backlog_Start.PRE)MUL(rHMI_RightPrime_Backlog_Stop_Time_S,1000,tRightPrime_Backlog_Stop.PRE);
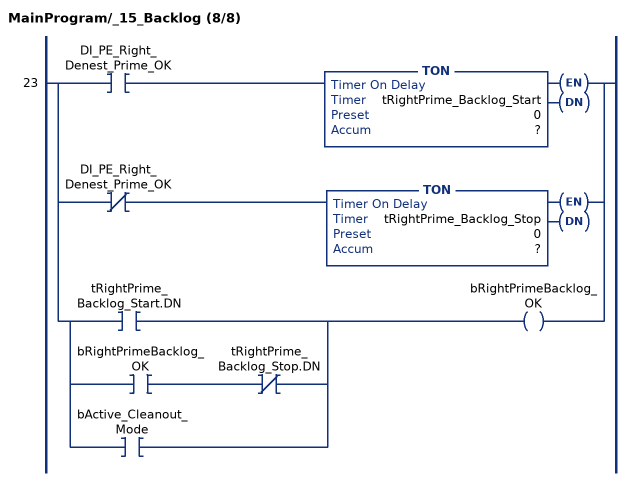
   23: [XIC(DI_PE_Right_Denest_Prime_OK) TON(tRightPrime_Backlog_Start,?,?) ,XIO(DI_PE_Right_Denest_Prime_OK) TON(tRightPrime_Backlog_Stop,?,?) ,[XIC(tRightPrime_Backlog_Start.DN) ,XIC(bRightPrimeBacklog_OK) XIO(tRightPrime_Backlog_Stop.DN) ,XIC(bActive_Cleanout_Mode) ] OTE(bRightPrimeBacklog_OK) ];
END_ROUTINE
